// TIA Portal V17 export
// export: Created 2024-08-20T13:26:12.0660753Z, ExportSetting WithDefaults, DisplayName Totally Integrated Automation Portal, DisplayVersion V17 Update 4, DisplayName TIA Portal Openness, DisplayVersion V17 Update 4, DisplayName TIA Portal Version Control Interface, DisplayVersion V17, DisplayName STEP 7 Professional, DisplayVersion V17 Update 4, DisplayName STEP 7 Safety, DisplayVersion V17, DisplayName WinCC Advanced, DisplayVersion V17 Update 4
DATA_BLOCK "INTPRO_DB"   // DB2
VERSION : 0.1
// stored: AutoNumber true, DBAccessibleFromOPCUA true, InstanceOfName INTPRO, InstanceOfType FB
"INTPRO"
   // VAR
   //    EE_P_NIV : Bool;
   //    EE_C1_NIV : Bool;
   //    EE_C2_NIV : Bool;
   //    EE_P_LS : Bool;
   //    EE_C1_LS : Bool;
   //    EE_C2_LS : Bool;
   //    HAB_P_EE : Bool;
   //    HAB_C1_EE : Bool;
   //    HAB_C2_EE : Bool;
   //    AUXP01 : Bool;
   //    BS01OK : Bool;
   //    BS02OK : Bool;
   //    BS03OK : Bool;
   //    L_BS01 : Bool;
   //    L_BS02 : Bool;
   //    L_BS03 : Bool;
   //    AUXP02 : Bool;
   //    AUXP03 : Bool;
   //    AUXP04 : Bool;
   //    AUXP05 : Bool;
   //    AUXP06 : Bool;
   //    AUXP07 : Bool;
   //    ETBS01_T001 : Int;
   //    ETBS02_T001 : Int;
   //    ETBS03_T001 : Int;
   //    BS01TO : Int;
   //    BS02TO : Int;
   //    BS03TO : Int;
   //    BS01TEOK : DInt;
   //    BS02TEOK : DInt;
   //    BS03TEOK : DInt;
   //    TE00 { S7_SetPoint := 'True'} : IEC_TIMER;
   //    RODEE { S7_SetPoint := 'True'} : "ROD4";
   // END_VAR
BEGIN
END_DATA_BLOCK
